(* PLC project LD_FB.project, Inovance company InoProShop(V1.8.1.3) InoProShop(V1.8.1.3) *)
(* stored: creationDateTime 2025-03-14T15:06:19.4890163, modificationDateTime 2025-03-13T22:41:36.6403457 *)

PROGRAM PLC_PRG
  VAR
    FB00 : FB0;
    tmp : INT;
    tot : INT;
    TON1 : TON;
  END_VAR
  VAR  (* added by the conversion: wires and edge detectors of the diagram *)
    _GT8_ENO : BOOL;
    _GT8_OUT : BOOL;
  END_VAR

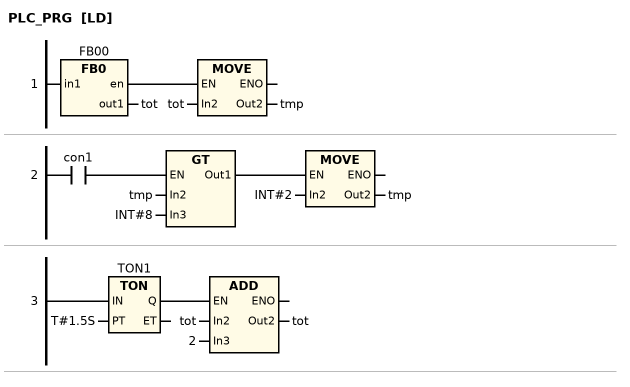
(* LD diagram, written out as Structured Text *)
(* 网络注释 *)

FB00(in1 := TRUE, out1 => tot);
IF FB00.en THEN tmp := tot; END_IF;
_GT8_OUT := GT(EN := con1, IN1 := tmp, IN2 := INT#8, ENO => _GT8_ENO);
IF _GT8_OUT THEN tmp := INT#2; END_IF;
(* 网络注释 *)

TON1(IN := TRUE, PT := T#1.5S);
IF TON1.Q THEN tot := tot + 2; END_IF;
END_PROGRAM

FUNCTION_BLOCK FB0
  VAR_INPUT
    in1 : BOOL;
  END_VAR
  VAR_OUTPUT
    out1 : INT;
    en : BOOL;
  END_VAR
  VAR
    TON0 : TON;
  END_VAR

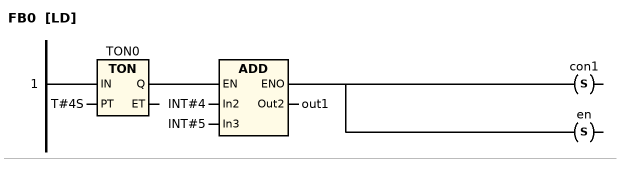
(* LD diagram, written out as Structured Text *)
(* 网络注释 *)

TON0(IN := TRUE, PT := T#4S);
IF TON0.Q THEN out1 := INT#4 + INT#5; END_IF;
IF TON0.Q THEN con1 := TRUE; END_IF;
IF TON0.Q THEN en := TRUE; END_IF;
END_FUNCTION_BLOCK

CONFIGURATION Application
  RESOURCE Application ON PLC
    VAR_GLOBAL RETAIN PERSISTENT  (* GVL *)
      con1 AT %MB131072 : BOOL := TRUE;
      con2 : BOOL := TRUE;
      norm1 : INT;
    END_VAR
  END_RESOURCE
END_CONFIGURATION
